
FUNCTION CB_le_tod : BOOL


TITLE = ' Test Whether IN0 is lower than or equal to IN1 '
VERSION : '1.0'
AUTHOR  : CB
NAME    : le_tod
FAMILY  : TNI

VAR_INPUT
    IN0 : TOD;
    IN1 : TOD;
END_VAR

BEGIN

CB_le_tod := (IN0 <= IN1);

END_FUNCTION
